SUBAPPLICATION WhiteGreenPurpleBackground1_AX (* Hintergrundfarbe fuer 1 Objekt (AX-Adapter), 3 Zustaende: DI1=FALSE -> Weiss (nicht erfuellt), DI1=TRUE -> Gruen (erfuellt), DI2=TRUE -> Violett (Override, hat Vorrang vor DI1). Franz: Vorbedingungs-Badges (Saege/Baender/Zapfwelle) bei Aufnahme-Automatik. *)
  (* Standard: 61499-2; Description: Copyright (c) 2026 Meisterschulen am Ostbahnhof This program and the accompanying materials are made available under the terms of the Eclipse Public License 2.0 which is available at https://www.eclipse.org/legal/epl-2.0/ SPDX-License-Identifier: EPL-2.0 *)
  (* Version 1.0, 2026-10-01, Franz Höpfinger, Meisterschulen am Ostbahnhof, initial implementation, analog GreenWhiteBackground1_AX - 2 verschachtelte F_SEL (nicht AX_SEL, da ein einzelnes AX_SEL nur bei Aenderung des EIGENEN G neu auswertet und die 2. Stufe bei einer Aenderung von DI1 sonst nicht nachziehen wuerde) - beide F_SEL werden ueber einen gemeinsamen Trigger (E_MERGE_2 aus DI1.E1/DI2.E1) in Reihe neu ausgewertet, damit eine Aenderung von DI1 ODER DI2 immer die komplette, korrekte Farbe liefert. *)
  PACKAGE MyLib::sys;
  IMPORT isobus::UT::Q::const::IDs::ID_NULL;
  IMPORT isobus::UT::Q::const::colours::COLOR_GREEN;
  IMPORT isobus::UT::Q::const::colours::COLOR_WHITE;
  IMPORT isobus::UT::Q::const::colours::COLOR_PURPLE;
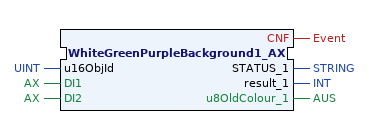
  EVENT_OUTPUT
    CNF; (* Execution Confirmation *)
  END_EVENT
  VAR_INPUT
    u16ObjId : UINT := ID_NULL; (* Object ID Softkey/Button/OutputText *)
  END_VAR
  VAR_OUTPUT
    STATUS_1 : STRING; (* Service Status *)
    result_1 : INT; (* retval see description *)
  END_VAR
  SOCKETS
    DI1 : adapter::types::unidirectional::AX; (* Bedingung erfuellt (FALSE=Weiss, TRUE=Gruen) - ohne Vorrang, siehe DI2 *)
    DI2 : adapter::types::unidirectional::AX; (* Override aktiv (TRUE=Violett) - hat Vorrang vor DI1 *)
  END_SOCKETS
  PLUGS
    u8OldColour_1 : adapter::types::unidirectional::AUS; (* Old value of color *)
  END_PLUGS
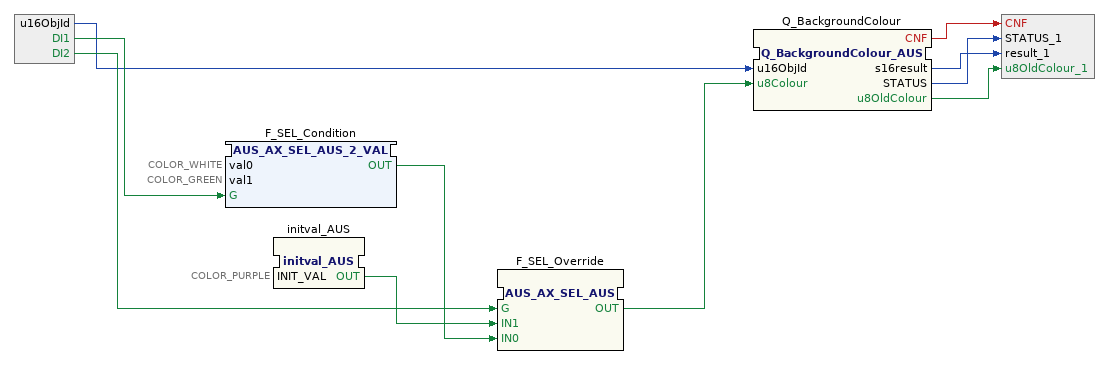
  FBS
    Q_BackgroundColour : isobus::UT::Q::Q_BackgroundColour_AUS;
    F_SEL_Override : adapter::iec61131::selection::AUS_AX_SEL_AUS;
    initval_AUS : adapter::types::unidirectional::AUS::initval::initval_AUS(INIT_VAL := COLOR_PURPLE);
  END_FBS
  SUBAPPS
    F_SEL_Condition : MyLib::sys::AUS_AX_SEL_AUS_2_VAL(val0 := COLOR_WHITE, val1 := COLOR_GREEN);
  END_SUBAPPS
  EVENT_CONNECTIONS
    Q_BackgroundColour.CNF TO CNF;
  END_CONNECTIONS
  DATA_CONNECTIONS
    u16ObjId TO Q_BackgroundColour.u16ObjId;
    Q_BackgroundColour.s16result TO result_1;
    Q_BackgroundColour.STATUS TO STATUS_1;
  END_CONNECTIONS
  ADAPTER_CONNECTIONS
    DI2 TO F_SEL_Override.G;
    DI1 TO F_SEL_Condition.G;
    Q_BackgroundColour.u8OldColour TO u8OldColour_1;
    F_SEL_Override.OUT TO Q_BackgroundColour.u8Colour;
    initval_AUS.OUT TO F_SEL_Override.IN1;
    F_SEL_Condition.OUT TO F_SEL_Override.IN0;
  END_CONNECTIONS
END_SUBAPPLICATION
